(* Logix 5000 project; controller DispersionPlc vendor 1 type 14 code 108 rev 34.11; software revision 34.01 *)

TASK MainTask (continuous, watchdog 500 ms) : MainProgram, Unit_K400, Unit_V4307, Unit_V4306, Unit_T4302, Unit_S4352, Unit_S51, Unit_RO_HE4305, Simulation, General_Purpose, Deviation_Alarms, Unit_K200
TASK Periodic_100ms (periodic, rate 100 ms, priority 2, watchdog 500 ms) : PIDLoops

MODULES
   Local : vendor 1 type 14 code 108 (Compact 0, rev 34.11)
      Input_2 : vendor 1 type 7 code 82 (Compact 3, rev 1.1, Input RPI 2 ms)
      Input_1 : vendor 1 type 7 code 82 (Compact 2, rev 1.1, Input RPI 2 ms)
      Input_3 : vendor 1 type 7 code 82 (Compact 4, rev 1.1, Input RPI 2 ms)
      Therm_1 : vendor 1 type 10 code 36 (Compact 8, rev 1.2, Input RPI 2 ms)
      IF81 : 1769-MODULE (Compact 12, rev 1.1, Output RPI 2 ms)
      AnaOut : vendor 1 type 10 code 40 (Compact 13, rev 2.1, Output RPI 2 ms)
      Therm_3 : vendor 1 type 10 code 36 (Compact 10, rev 1.2, Input RPI 2 ms)
      Sdn : vendor 1 type 12 code 105 (Compact 1, rev 2.1, Output RPI 2 ms)
      IF8 : 1769-MODULE (Compact 11, rev 1.1, Output RPI 2 ms)
      Output_1 : 1769-OW16 (Compact 5, rev 1.1, Output RPI 2 ms)
      Output_2 : 1769-OW16 (Compact 6, rev 1.1, Output RPI 2 ms)
      Output_3 : 1769-OW16 (Compact 7, rev 1.1, Output RPI 2 ms)
      Therm_2 : vendor 1 type 10 code 36 (Compact 9, rev 1.2, Input RPI 2 ms)
      AG_4306 : PowerFlex 525-EENET (Ethernet 10.61.51.161, rev 5.1, Output RPI 20 ms)
      P_4302_2 : PowerFlex 525-EENET (Ethernet 10.61.51.163, rev 5.1, Output RPI 20 ms)
      AG_4302 : vendor 1 type 142 code 1168 (Ethernet 10.61.51.160, rev 9.1, Output RPI 20 ms)
          : vendor 1 type 142 code 57760 (RhinoBP 5, rev 1.1)
          : vendor 1 type 142 code 33184 (RhinoBP 14, rev 2.5)
      AG_4307 : PowerFlex 525-EENET (Ethernet 10.61.51.162, rev 5.1, Output RPI 20 ms)
      New_INX_IO : vendor 1 type 12 code 298 (Ethernet 10.61.51.115, rev 1.1)
         AC_Inputs : vendor 1 type 7 code 82 (Compact 1, rev 3.1, Input RPI 100 ms)
         Digital_Inputs : 1769-IQ16 (Compact 5, rev 1.1, Input RPI 20 ms)
         Relay_Outputs : 1769-OW8I (Compact 2, rev 3.1, Output RPI 100 ms)
         Analog_Inputs : vendor 1 type 10 code 44 (Compact 3, rev 2.1, Output RPI 100 ms)
         Analog_Outputs : vendor 1 type 10 code 40 (Compact 4, rev 2.2, Output RPI 100 ms)
         Digital_Outputs : 1769-OB16 (Compact 6, rev 2.1, Output RPI 20 ms)
      RIO1_Rack1 : vendor 1 type 12 code 298 (Ethernet 10.61.51.164, rev 1.1)
         DIn : vendor 1 type 7 code 82 (Compact 3, rev 1.1, Input RPI 20 ms)
         DOut : 1769-OW16 (Compact 4, rev 1.1, Output RPI 20 ms)
         AOut : vendor 1 type 10 code 40 (Compact 2, rev 2.1, Output RPI 80 ms)
         AIn : 1769-IF8 (Compact 1, rev 1.1, Output RPI 80 ms)
END_MODULES

TYPE Alarm_SPT :
STRUCT
   HIHI : REAL;
   HI : REAL;
   LO : REAL;
   LOLO : REAL;
END_STRUCT
END_TYPE

TYPE AStd_AnalogAlarm :
STRUCT
   AckC : BOOL;
   LatchA : BOOL;
   DetectS : BOOL;
   BitS : BOOL;
   InhibitC : BOOL;
   LimitC : REAL;
   LimitOffSetC : REAL;
   Tmr : TIMER;
   Disabled : BOOL;
END_STRUCT
END_TYPE

TYPE AStd_AnalogInput :
STRUCT
   Raw : REAL;
   AckAreaC : BOOL;
   AckC : BOOL;
   Scaled : REAL;
   Scaling : AStd_AnalogScaling;
   LowLow : AStd_AnalogAlarm;
   Low : AStd_AnalogAlarm;
   High : AStd_AnalogAlarm;
   HighHigh : AStd_AnalogAlarm;
   Fault : AStd_AnalogAlarm;
   FaultReset : REAL;
END_STRUCT
END_TYPE

TYPE AStd_AnalogOutput :
STRUCT
   Scaled : REAL;
   Raw : REAL;
   Scaling : AStd_AnalogScaling;
END_STRUCT
END_TYPE

TYPE AStd_AnalogScaling :
STRUCT
   RawMinS : REAL;
   RawMaxS : REAL;
   EngMinS : REAL;
   EngMaxS : REAL;
END_STRUCT
END_TYPE

TYPE AStd_DateTimeFormat :
STRUCT
   CurrentYear : DINT;
   CurrentMonth : DINT;
   CurrentDay : DINT;
   CurrentHour : DINT;
   CurrentMinute : DINT;
   CurrentSecond : DINT;
   DateTimeBuild : STRING;
   TemporaryString : STRING;
   DateTimeBuffer : DINT[10];
   ConstantZero : STRING;
   ConstantColon : STRING;
   ConstantDash : STRING;
   ConstantSpace : STRING;
   CurrentDateTime : STRING;
   SetTimeC : BOOL;
END_STRUCT
END_TYPE

TYPE AStd_Device_Perm :
STRUCT
   InterlockS : DINT;
   SafetyS : DINT;
   IntlkS : BOOL;
   SafeS : BOOL;
   InterlockInhibitC : DINT;
   SafetyInhibitC : DINT;
   IntSafDisp : DINT;
   InterlockTimers : TimerArray;
END_STRUCT
END_TYPE

TYPE AStd_DiscreteAlarm :
STRUCT
   AckC : BOOL;
   LatchA : BOOL;
   DetectS : BOOL;
   BitS : BOOL;
   InhibitC : BOOL;
   Tmr : TIMER;
END_STRUCT
END_TYPE

TYPE AStd_DiscreteInput :
STRUCT
   InI : BOOL;
   Alm : AStd_DiscreteAlarm;
END_STRUCT
END_TYPE

TYPE AStd_FVNR :
STRUCT
   AutoC : BOOL;
   ManC : BOOL;
   AutoS : BOOL;
   StartC : BOOL;
   StopC : BOOL;
   RunO : BOOL;
   RunI : BOOL;
   DiscI : BOOL;
   AlmS : BOOL;
   RuntimeResetC : BOOL;
   AutoCtrlS : BOOL;
   AutoCtrlC : DINT;
   RuntimeS : DINT;
   Perm : AStd_Device_Perm;
   MiscAlm : AStd_DiscreteAlarm;
   DiscAlm : AStd_DiscreteAlarm;
   AckC : BOOL;
END_STRUCT
END_TYPE

TYPE AStd_GeneralPurp :
STRUCT
   AlwaysOff : BOOL;
   AlwaysOn : BOOL;
   FirstScan : BOOL;
   PowerUpDelay : BOOL;
   AlternateScan : BOOL;
   HalfSecondPulse : BOOL;
   HalfSecondSquare : BOOL;
   OneSecondPulse : BOOL;
   OneSecondSquare : BOOL;
   PowerUpDelayOS : BOOL;
   Tmr : TIMER[5];
   ONS : DINT;
END_STRUCT
END_TYPE

TYPE AStd_PIDInterface :
STRUCT
   AutoC : BOOL;
   ManC : BOOL;
   AutoS : BOOL;
   AutoCtrlC : DINT;
   AutoCtrlS : BOOL;
   EnableS : BOOL;
   ManOut : REAL;
   SPC : REAL;
   PGainC : REAL;
   IGainC : REAL;
   DGainC : REAL;
   PGainS : REAL;
   IGainS : REAL;
   DGainS : REAL;
   SPS : REAL;
   PVS : REAL;
   CVS : REAL;
   Perm : AStd_Device_Perm;
END_STRUCT
END_TYPE

TYPE AStd_PLCStatus :
STRUCT
   ForcePresent : BOOL;
   BatteryFault : BOOL;
   MinorFaultBits : DINT;
   ForceStatus : DINT;
   PLCScanTime : REAL;
   PLCScanTimeMin : REAL;
   CodeVersion : STRING;
   DateTime : AStd_DateTimeFormat;
   PLCForcePresent : AStd_DiscreteAlarm;
   PLCBatteryFault : AStd_DiscreteAlarm;
   PLCPowerUp : AStd_DiscreteAlarm;
END_STRUCT
END_TYPE

TYPE AStd_PLI :
STRUCT
   StartC : BOOL;
   HoldC : BOOL;
   RestartC : BOOL;
   AbortC : BOOL;
   CompleteC : BOOL;
   ResetC : BOOL;
   UserStopC : BOOL;
   IdleS : BOOL;
   RunS : BOOL;
   HeldS : BOOL;
   AbortS : BOOL;
   DoneS : BOOL;
   CurrentStateCodeS : DINT;
   PreventStartS : DINT;
   AlarmS : DINT;
   Adv : BOOL;
   StepNo : DINT;
   StepBit : DINT;
   ONS : DINT;
   UnitProc_ActiveS : BOOL;
   UnitProc_RecipePointerS : DINT;
   UnitProc_PhaseID : DINT;
   RealParameters : REAL[20];
   BoolParameters : BOOL[32];
   DINTParameters : DINT[20];
   PreventStartInhibitC : DINT;
   AlarmInhibitC : DINT;
   IntSafDisp : DINT;
   InterlockTimers : TimerArray;
END_STRUCT
END_TYPE

TYPE AStd_VFD :
STRUCT
   AutoC : BOOL;
   ManC : BOOL;
   AutoS : BOOL;
   StartC : BOOL;
   StartRevC : BOOL;
   StopC : BOOL;
   ManSpdC : REAL;
   AutoSpdC : REAL[10];
   AutoSpdS : REAL;
   SpeedI : AStd_AnalogInput;
   SpeedC : AStd_AnalogOutput;
   AutoCtrlC : DINT;
   AutoRevCtrlC : DINT;
   AutoCtrlS : BOOL;
   AutoRevCtrlS : BOOL;
   RunI : BOOL;
   DiscI : BOOL;
   DriveFltI : BOOL;
   RunTimeResetC : BOOL;
   RunTimeS : DINT;
   RunO : BOOL;
   ReverseS : BOOL;
   AckC : BOOL;
   AckAreaC : BOOL;
   Perm : AStd_Device_Perm;
   MiscAlm : AStd_DiscreteAlarm;
   DiscAlm : AStd_DiscreteAlarm;
   DriveFlt : AStd_DiscreteAlarm;
   AlmS : BOOL;
END_STRUCT
END_TYPE

TYPE AStd_VlvModulating :
STRUCT
   AutoC : BOOL;
   ManC : BOOL;
   AutoS : BOOL;
   OpenC : BOOL;
   CloseC : BOOL;
   AutoCtrlS : BOOL;
   Perm : AStd_Device_Perm;
   ManPosC : REAL;
   AutoCtrlC : DINT;
   AutoPosC : REAL[10];
   AutoPosS : REAL;
   ScaledO : REAL;
   Scaling : AStd_AnalogScaling;
   RawO : REAL;
END_STRUCT
END_TYPE

TYPE AStd_VlvOC :
STRUCT
   AutoC : BOOL;
   ManC : BOOL;
   AutoS : BOOL;
   OpenC : BOOL;
   CloseC : BOOL;
   StopC : BOOL;
   OpenO : BOOL;
   CloseO : BOOL;
   OpenI : BOOL;
   ClosedI : BOOL;
   CycleCountResetC : BOOL;
   AlmS : BOOL;
   AutoCtrlS : BOOL;
   AckC : BOOL;
   AckAreaC : BOOL;
   cfgHasZSC : BOOL;
   cfgHasZSO : BOOL;
   AutoCtrlC : DINT;
   CycleCountS : DINT;
   Perm : AStd_Device_Perm;
   MiscAlm : AStd_DiscreteAlarm;
END_STRUCT
END_TYPE

TYPE bit64 :
STRUCT
   Bit : BOOL[64];
END_STRUCT
END_TYPE

TYPE Kettle :
STRUCT
   Level : Proc_Var;
   Heating : Proc_Var;
   Pressure : Proc_Var;
   Cooling : Proc_Var;
   Combined : Proc_Var;
   Auto_Manual : BOOL;
   Heat_Manual_Output_Request : REAL;
   ValveOutput : INT;
   CoolingValveOutput : INT;
   ValvePercOpen : REAL;
   OverheadTemp : REAL;
   H20SupplyValvePercOpen : REAL;
   H20SupplyValveOutput : INT;
   RupDiscRelfTemp : REAL;
   Zone1ActuatedValvePos : BOOL;
   Zone2ActuatedValvePos : BOOL;
   Zone3ActuatedValvePos : BOOL;
   Cool_Auto_Manual : BOOL;
   Cool_Manual_Output_Request : REAL;
   BatchStart : BOOL;
   BatchRunning : BOOL;
   BatchID : STRING;
   ProductID : STRING;
   Proportional : REAL;
   Integral : REAL;
   Derivative : REAL;
   Timer : TIMER[5];
   BatchStop : BOOL;
   Alarm : BOOL;
   Cooling_Valve_Status : BOOL;
   Reflux : BOOL;
   BIts : DINT;
   Operation : DINT;
END_STRUCT
END_TYPE

TYPE Proc_Var :
STRUCT
   Value_Name : STRING;
   Value_Raw : INT;
   Value : REAL;
   Volume_Value : REAL;
   Setpoint : REAL;
   Error_Val : REAL;
   MMI_Level : REAL;
   Value_Sf : REAL;
   Volume_Sf : REAL;
   Offset : REAL;
   HIHI : REAL;
   HI : REAL;
   LO : REAL;
   LOLO : REAL;
   OUT : REAL;
   HIHI_ALM : BOOL;
   HI_ALM : BOOL;
   LO_ALM : BOOL;
   LOLO_ALM : BOOL;
   High_Limit_Switch : BOOL;
   Lo_Limit_Switch : BOOL;
   LossOfInput : BOOL;
END_STRUCT
END_TYPE

TYPE Seq64 :
STRUCT
   Val : DINT;
   Ret : DINT;
   Tmr : TIMER[64];
   probit : BOOL[64];
   Ons : BOOL[64];
   seqstrings : STRING[64];
   alarmstrings : STRING[64];
   seqstring : STRING;
   alarmstring : STRING;
   Alarm_Timers : TIMER[64];
   Alarm_Scanner : DINT;
   Alarm_Display_Index : DINT;
   Alarm_Display_Que : DINT;
   ClearAlarms : BOOL;
   Active : BOOL;
   Sq : Stp64;
   MANUAL : bit64;
   Alarm : bit64;
   ALARM_TIMER : TIMER;
   ALARM_DISPLAY : DINT;
   AutoMode : BOOL;
   ManualMode : BOOL;
   AutoManualPb : BOOL;
   ClearAlarmTmr : TIMER;
   HMI : bit64;
   VAL_HOLD : DINT;
   CLEAR_SEQ : BOOL;
   AlarmHist : bit64;
   AlarmHistEnable : bit64;
   AlarmONS : bit64;
   AlarmHistString : STRING;
   Alarm_Setpoint : Alarm_SPT;
END_STRUCT
END_TYPE

TYPE Stp64 :
STRUCT
   Step : BOOL[64];
   Dn : BOOL[64];
END_STRUCT
END_TYPE

TYPE TimerArray :
STRUCT
   Timers : TIMER[10];
END_STRUCT
END_TYPE

TYPE Udt_Tank :
STRUCT
   Name : STRING;
   Level : Proc_Var;
   Temperature : Proc_Var;
   Pressure : Proc_Var;
   PercentChange : REAL;
   MaxPercentChange : BOOL;
   LvlSampleAtPmpStart : REAL;
   Enabled : BOOL;
   MaxPercChangeAlr : BOOL;
   Number : INT;
END_STRUCT
END_TYPE

TYPE VFD :
STRUCT
   TargetDriveSpeed : INT;
   I_Ready : BOOL;
   I_Running : BOOL;
   I_CmdDir : BOOL;
   I_ActDir : BOOL;
   I_Accelerating : BOOL;
   I_Decelerating : BOOL;
   I_Alarm : BOOL;
   I_Fault : BOOL;
   I_AtSpeed : BOOL;
   I_LocalContStat1 : BOOL;
   I_LocalContStat2 : BOOL;
   I_LocalContStat3 : BOOL;
   I_Refferance1 : BOOL;
   I_Refferance2 : BOOL;
   I_Refferance3 : BOOL;
   I_Refferance4 : BOOL;
   I_V_Units_Fb : REAL;
   I_Act_Amps : REAL;
   I_DatalinkA2_Fb : REAL;
   O_Stop : BOOL;
   O_Run : BOOL;
   O_Jog : BOOL;
   O_ClrFlts : BOOL;
   O_DirBit1 : BOOL;
   O_DirBit2 : BOOL;
   O_LocalContol : BOOL;
   O_MopInc : BOOL;
   O_MOP_Accel1 : BOOL;
   O_Accel2 : BOOL;
   O_MOP_Decel1 : BOOL;
   O_MOP_Decel2 : BOOL;
   O_Reff_Sel1 : BOOL;
   O_Reff_Sel2 : BOOL;
   O_Reff_Sel3 : BOOL;
   O_V_CmdReff : REAL;
   O_Dlnk_A1_Reff : INT;
   O_Dlnk_A2_Reff : INT;
   SpeedScaleIn : REAL;
   SpeedScaleOut : REAL;
   MaxOutPut : REAL;
   MinOutput : REAL;
   DriveSpeedReff : REAL;
END_STRUCT
END_TYPE

ADD_ON_INSTRUCTION Analog_Scale   (* revision 1.0, vendor DM *)
VAR_INPUT
   Analog_In : REAL; {required}
   Offset_In : REAL; {required}
   Analog_Min_In : REAL; {required}
   Analog_Max_In : REAL; {required}
   Analog_Min_Out : REAL; {required}
   Analog_Max_Out : REAL; {required}
END_VAR
VAR_OUTPUT
   Analog_Out : REAL; {access Read Only, required}
END_VAR
VAR_INPUT
   Offset_Out : REAL; {required}
END_VAR
VAR
   F8 : REAL[10];
END_VAR

ROUTINE Logic   (* ladder *)
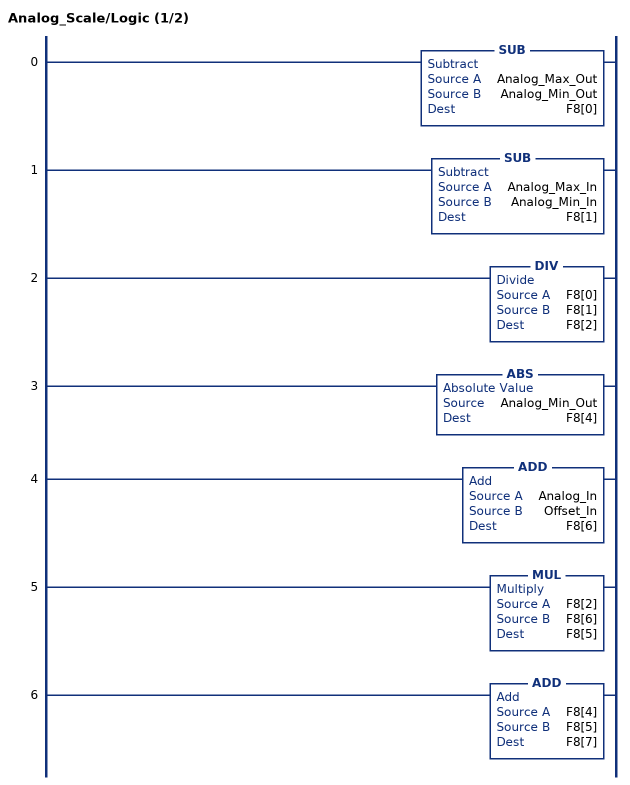
   0: SUB(Analog_Max_Out,Analog_Min_Out,F8[0]);
   1: SUB(Analog_Max_In,Analog_Min_In,F8[1]);
   2: DIV(F8[0],F8[1],F8[2]);
   3: ABS(Analog_Min_Out,F8[4]);
   4: ADD(Analog_In,Offset_In,F8[6]);
   5: MUL(F8[2],F8[6],F8[5]);
   6: ADD(F8[4],F8[5],F8[7]);
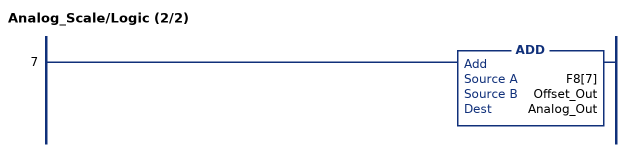
   7: ADD(F8[7],Offset_Out,Analog_Out);
END_ROUTINE
END_ADD_ON_INSTRUCTION

ADD_ON_INSTRUCTION AOI_Toggle   (* revision 1.0, vendor Danieli Taranis, ExecutePrescan, ExecuteEnableInFalse *)
VAR_OUTPUT
   Q : BOOL; {visible}
   QNot : BOOL; {visible}
END_VAR
VAR
   StorageBit : BOOL; {access None}
   RunOnce : BOOL; {access None}
END_VAR

ROUTINE EnableInFalse   (* structured text *)
   RunOnce:=0;
END_ROUTINE

ROUTINE Logic   (* structured text *)
   //Perform one shot logic and
   //then evaluate the state of Q.
   //
   //Flip value of Q to opposite value.
   //Set QNot to opposite of Q
   //Store internal RunOnce for one shot logic
   
   IF NOT RunOnce THEN
   
   	Q:=NOT Q;
   	QNot:=NOT Q;
   	RunOnce:=1;
   
   END_IF;
   
   
   
   
END_ROUTINE

ROUTINE Prescan   (* structured text *)
   Q:=0;
   RunOnce:=0;
   
END_ROUTINE
END_ADD_ON_INSTRUCTION

ADD_ON_INSTRUCTION AStd_AI_AOI   (* revision 1.0, vendor Avanceon *)
VAR_IN_OUT
   AnalogInput : AStd_AnalogInput; {required}
END_VAR
VAR_INPUT
   InputRaw_I : REAL; {required}
   cfgRawMin : REAL := 4000.0; {required}
   cfgRawMax : REAL := 20000.0; {required}
   cfgEUMin : REAL; {required}
   cfgEUMax : REAL := 100.0; {required}
END_VAR
VAR_OUTPUT
   Scaled : REAL; {access Read Only, visible}
END_VAR
VAR_INPUT
   CommsStatus : BOOL; {required}
END_VAR

ROUTINE Logic   (* ladder *)
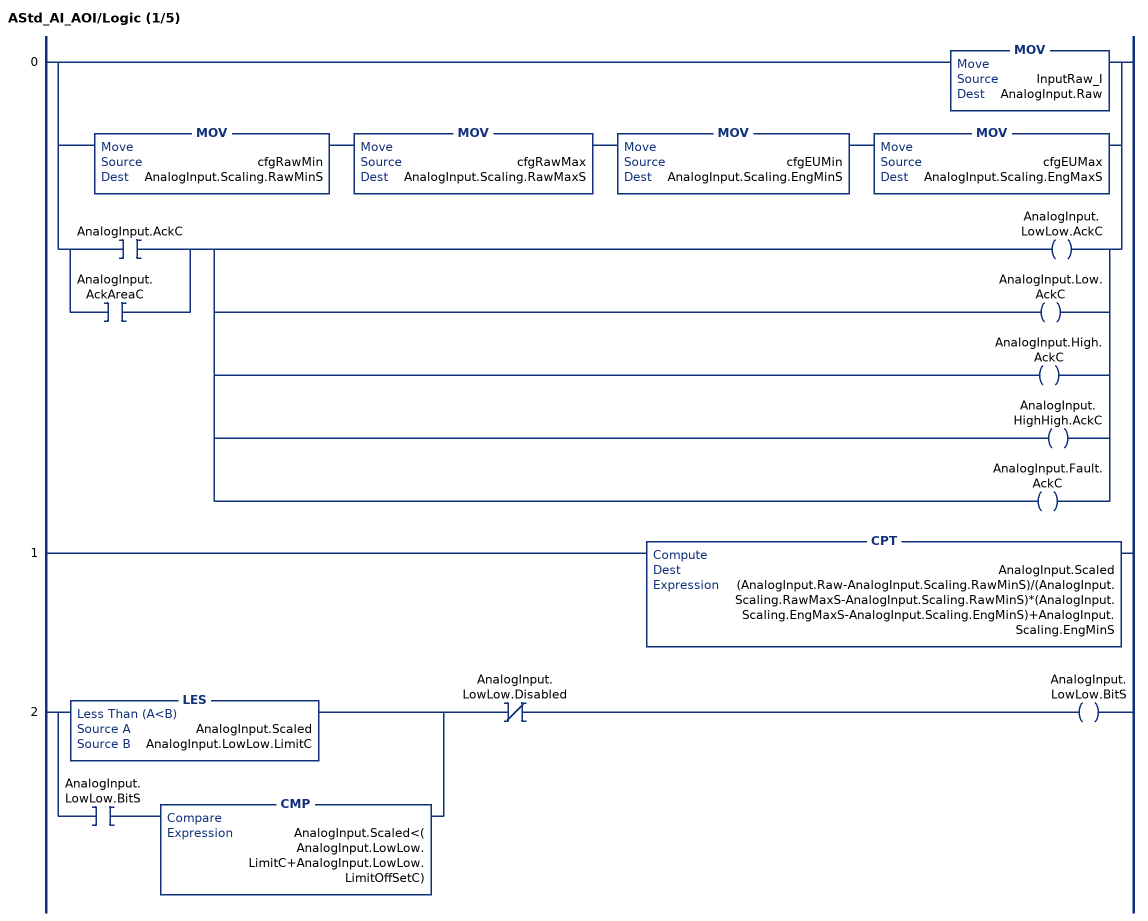
   0: [MOV(InputRaw_I,AnalogInput.Raw) ,MOV(cfgRawMin,AnalogInput.Scaling.RawMinS) MOV(cfgRawMax,AnalogInput.Scaling.RawMaxS) MOV(cfgEUMin,AnalogInput.Scaling.EngMinS) MOV(cfgEUMax,AnalogInput.Scaling.EngMaxS) ,[XIC(AnalogInput.AckC) ,XIC(AnalogInput.AckAreaC) ] [OTE(AnalogInput.LowLow.AckC) ,OTE(AnalogInput.Low.AckC) ,OTE(AnalogInput.High.AckC) ,OTE(AnalogInput.HighHigh.AckC) ,OTE(AnalogInput.Fault.AckC) ] ];
   1: CPT(AnalogInput.Scaled,(AnalogInput.Raw-AnalogInput.Scaling.RawMinS)/(AnalogInput.Scaling.RawMaxS-AnalogInput.Scaling.RawMinS)*(AnalogInput.Scaling.EngMaxS-AnalogInput.Scaling.EngMinS)+AnalogInput.Scaling.EngMinS);
   2: [LES(AnalogInput.Scaled,AnalogInput.LowLow.LimitC) ,XIC(AnalogInput.LowLow.BitS) CMP(AnalogInput.Scaled<(AnalogInput.LowLow.LimitC+AnalogInput.LowLow.LimitOffSetC)) ]XIO(AnalogInput.LowLow.Disabled)OTE(AnalogInput.LowLow.BitS);
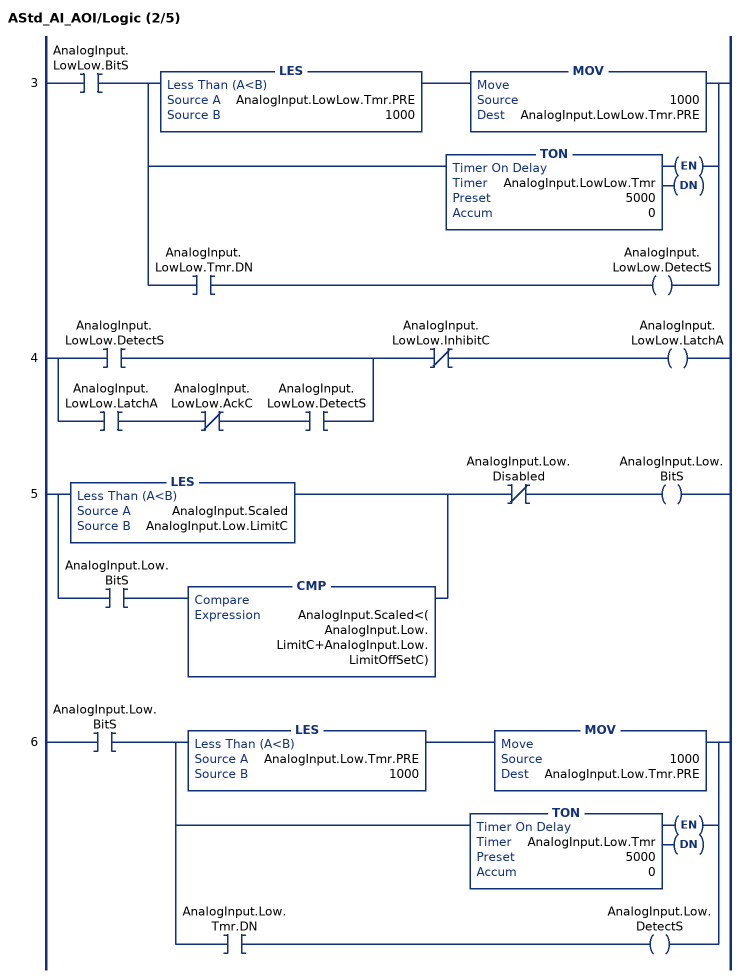
   3: XIC(AnalogInput.LowLow.BitS)[LES(AnalogInput.LowLow.Tmr.PRE,1000) MOV(1000,AnalogInput.LowLow.Tmr.PRE) ,TON(AnalogInput.LowLow.Tmr,5000,0) ,XIC(AnalogInput.LowLow.Tmr.DN) OTE(AnalogInput.LowLow.DetectS) ];
   4: [XIC(AnalogInput.LowLow.DetectS) ,XIC(AnalogInput.LowLow.LatchA) XIO(AnalogInput.LowLow.AckC) XIC(AnalogInput.LowLow.DetectS) ]XIO(AnalogInput.LowLow.InhibitC)OTE(AnalogInput.LowLow.LatchA);
   5: [LES(AnalogInput.Scaled,AnalogInput.Low.LimitC) ,XIC(AnalogInput.Low.BitS) CMP(AnalogInput.Scaled<(AnalogInput.Low.LimitC+AnalogInput.Low.LimitOffSetC)) ]XIO(AnalogInput.Low.Disabled)OTE(AnalogInput.Low.BitS);
   6: XIC(AnalogInput.Low.BitS)[LES(AnalogInput.Low.Tmr.PRE,1000) MOV(1000,AnalogInput.Low.Tmr.PRE) ,TON(AnalogInput.Low.Tmr,5000,0) ,XIC(AnalogInput.Low.Tmr.DN) OTE(AnalogInput.Low.DetectS) ];
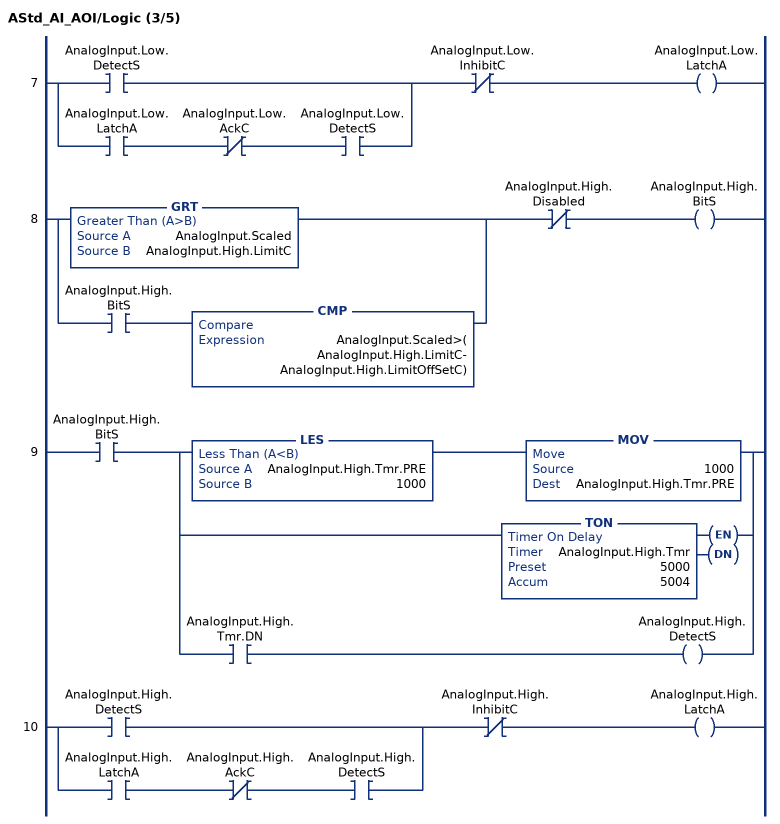
   7: [XIC(AnalogInput.Low.DetectS) ,XIC(AnalogInput.Low.LatchA) XIO(AnalogInput.Low.AckC) XIC(AnalogInput.Low.DetectS) ]XIO(AnalogInput.Low.InhibitC)OTE(AnalogInput.Low.LatchA);
   8: [GRT(AnalogInput.Scaled,AnalogInput.High.LimitC) ,XIC(AnalogInput.High.BitS) CMP(AnalogInput.Scaled>(AnalogInput.High.LimitC-AnalogInput.High.LimitOffSetC)) ]XIO(AnalogInput.High.Disabled)OTE(AnalogInput.High.BitS);
   9: XIC(AnalogInput.High.BitS)[LES(AnalogInput.High.Tmr.PRE,1000) MOV(1000,AnalogInput.High.Tmr.PRE) ,TON(AnalogInput.High.Tmr,5000,5004) ,XIC(AnalogInput.High.Tmr.DN) OTE(AnalogInput.High.DetectS) ];
   10: [XIC(AnalogInput.High.DetectS) ,XIC(AnalogInput.High.LatchA) XIO(AnalogInput.High.AckC) XIC(AnalogInput.High.DetectS) ]XIO(AnalogInput.High.InhibitC)OTE(AnalogInput.High.LatchA);
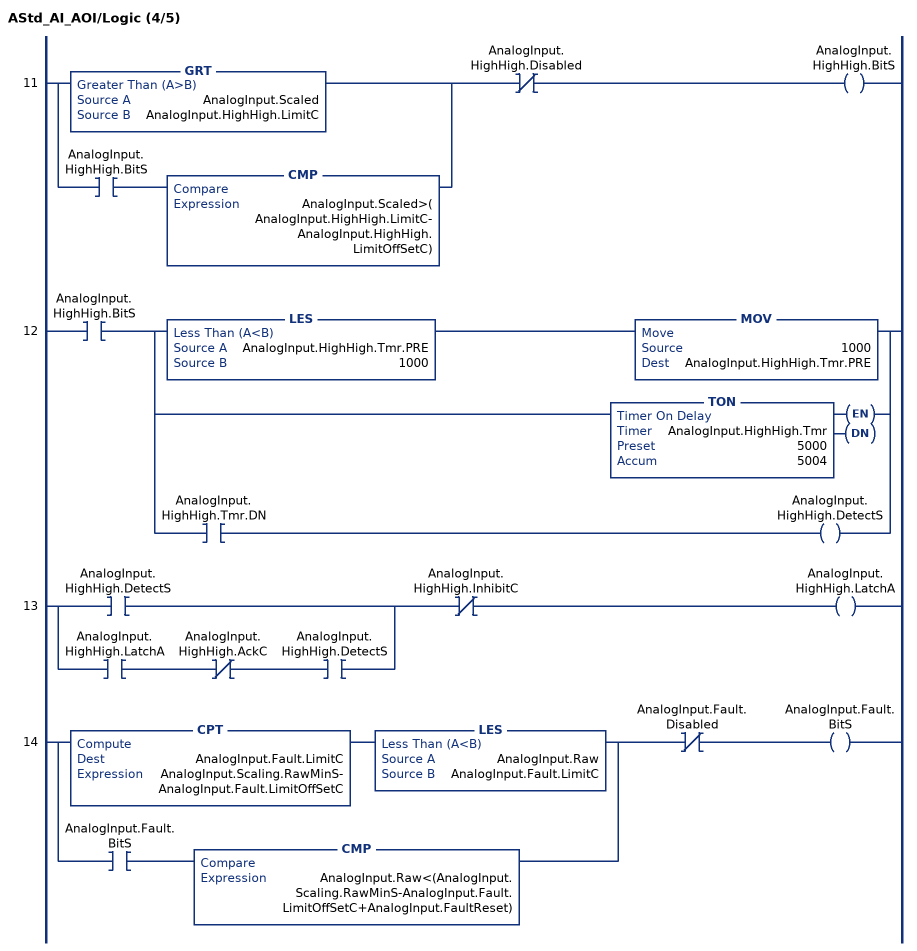
   11: [GRT(AnalogInput.Scaled,AnalogInput.HighHigh.LimitC) ,XIC(AnalogInput.HighHigh.BitS) CMP(AnalogInput.Scaled>(AnalogInput.HighHigh.LimitC-AnalogInput.HighHigh.LimitOffSetC)) ]XIO(AnalogInput.HighHigh.Disabled)OTE(AnalogInput.HighHigh.BitS);
   12: XIC(AnalogInput.HighHigh.BitS)[LES(AnalogInput.HighHigh.Tmr.PRE,1000) MOV(1000,AnalogInput.HighHigh.Tmr.PRE) ,TON(AnalogInput.HighHigh.Tmr,5000,5004) ,XIC(AnalogInput.HighHigh.Tmr.DN) OTE(AnalogInput.HighHigh.DetectS) ];
   13: [XIC(AnalogInput.HighHigh.DetectS) ,XIC(AnalogInput.HighHigh.LatchA) XIO(AnalogInput.HighHigh.AckC) XIC(AnalogInput.HighHigh.DetectS) ]XIO(AnalogInput.HighHigh.InhibitC)OTE(AnalogInput.HighHigh.LatchA);
   14: [CPT(AnalogInput.Fault.LimitC,AnalogInput.Scaling.RawMinS-AnalogInput.Fault.LimitOffSetC) LES(AnalogInput.Raw,AnalogInput.Fault.LimitC) ,XIC(AnalogInput.Fault.BitS) CMP(AnalogInput.Raw<(AnalogInput.Scaling.RawMinS-AnalogInput.Fault.LimitOffSetC+AnalogInput.FaultReset)) ]XIO(AnalogInput.Fault.Disabled)OTE(AnalogInput.Fault.BitS);
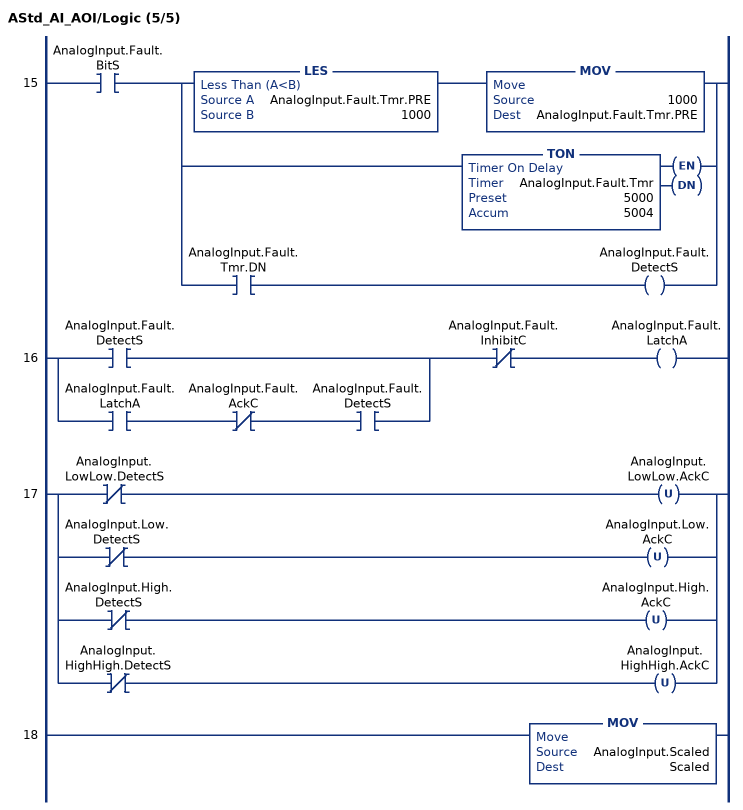
   15: XIC(AnalogInput.Fault.BitS)[LES(AnalogInput.Fault.Tmr.PRE,1000) MOV(1000,AnalogInput.Fault.Tmr.PRE) ,TON(AnalogInput.Fault.Tmr,5000,5004) ,XIC(AnalogInput.Fault.Tmr.DN) OTE(AnalogInput.Fault.DetectS) ];
   16: [XIC(AnalogInput.Fault.DetectS) ,XIC(AnalogInput.Fault.LatchA) XIO(AnalogInput.Fault.AckC) XIC(AnalogInput.Fault.DetectS) ]XIO(AnalogInput.Fault.InhibitC)OTE(AnalogInput.Fault.LatchA);
   17: [XIO(AnalogInput.LowLow.DetectS) OTU(AnalogInput.LowLow.AckC) ,XIO(AnalogInput.Low.DetectS) OTU(AnalogInput.Low.AckC) ,XIO(AnalogInput.High.DetectS) OTU(AnalogInput.High.AckC) ,XIO(AnalogInput.HighHigh.DetectS) OTU(AnalogInput.HighHigh.AckC) ];
   18: MOV(AnalogInput.Scaled,Scaled);
END_ROUTINE
END_ADD_ON_INSTRUCTION

ADD_ON_INSTRUCTION AStd_DI_AOI   (* revision 1.0, vendor Avanceon *)
VAR_IN_OUT
   DiscInputDevice : AStd_DiscreteInput; {required}
END_VAR
VAR_INPUT
   Input_I : BOOL; {access None, required}
   cfgFailSafe : BOOL; {access None, visible}
   cfgDebounceTmrPre : DINT := 1000; {access None, visible}
   cfgAlarmEnable : BOOL := 1; {access None, visible}
END_VAR
VAR_OUTPUT
   AlmS : BOOL; {access None, visible}
END_VAR
VAR
   Debounce : TIMER; {access None}
END_VAR

ROUTINE Logic   (* ladder *)
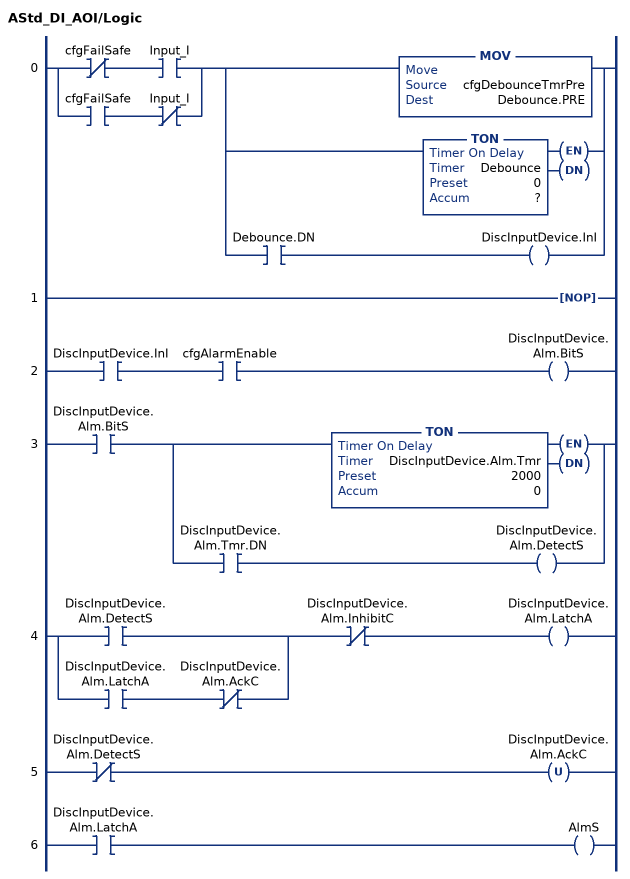
   0: [XIO(cfgFailSafe) XIC(Input_I) ,XIC(cfgFailSafe) XIO(Input_I) ][MOV(cfgDebounceTmrPre,Debounce.PRE) ,TON(Debounce,?,?) ,XIC(Debounce.DN) OTE(DiscInputDevice.InI) ];
   1: NOP();
   2: XIC(DiscInputDevice.InI)XIC(cfgAlarmEnable)OTE(DiscInputDevice.Alm.BitS);
   3: XIC(DiscInputDevice.Alm.BitS)[TON(DiscInputDevice.Alm.Tmr,2000,0) ,XIC(DiscInputDevice.Alm.Tmr.DN) OTE(DiscInputDevice.Alm.DetectS) ];
   4: [XIC(DiscInputDevice.Alm.DetectS) ,XIC(DiscInputDevice.Alm.LatchA) XIO(DiscInputDevice.Alm.AckC) ]XIO(DiscInputDevice.Alm.InhibitC)OTE(DiscInputDevice.Alm.LatchA);
   5: XIO(DiscInputDevice.Alm.DetectS)OTU(DiscInputDevice.Alm.AckC);
   6: XIC(DiscInputDevice.Alm.LatchA)OTE(AlmS);
END_ROUTINE
END_ADD_ON_INSTRUCTION

ADD_ON_INSTRUCTION AStd_FVNR_AOI   (* revision 1.0, vendor Avanceon *)
VAR_IN_OUT
   Motor : AStd_FVNR; {required}
END_VAR
VAR_INPUT
   AuxContact_I : BOOL; {required}
   Disconnect_I : BOOL; {required}
END_VAR
VAR_OUTPUT
   Coil_O : BOOL; {required}
END_VAR
VAR_INPUT
   cfgHasAUX : BOOL := 1; {access None, visible}
   cfgHasDISC : BOOL; {access None, visible}
END_VAR
VAR_OUTPUT
   AutoS : BOOL; {access Read Only, visible}
   RunS : BOOL; {access Read Only, visible}
   AlmS : BOOL; {access Read Only, visible}
END_VAR
VAR
   RuntimeHourTimer : TIMER := (PRE := 3600000); {access None}
END_VAR

ROUTINE Logic   (* ladder *)
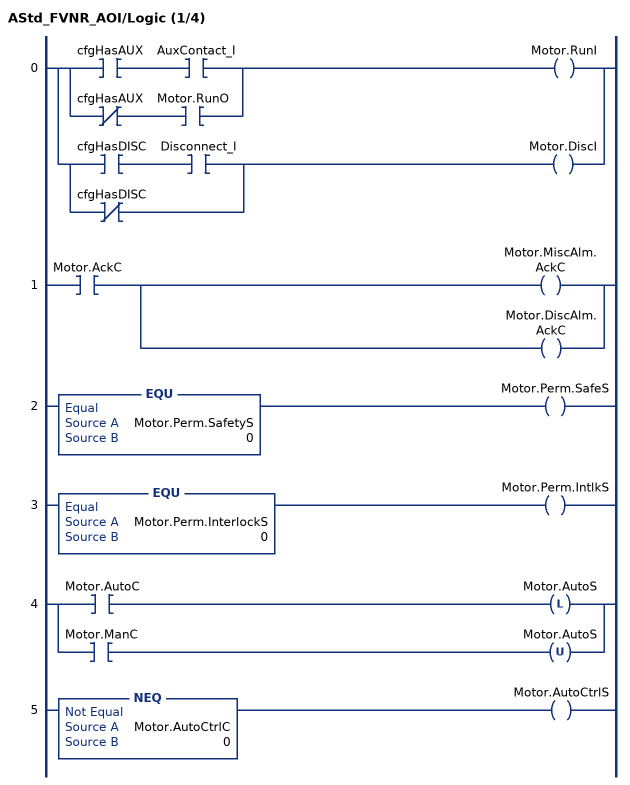
   0: [[XIC(cfgHasAUX) XIC(AuxContact_I) ,XIO(cfgHasAUX) XIC(Motor.RunO) ] OTE(Motor.RunI) ,[XIC(cfgHasDISC) XIC(Disconnect_I) ,XIO(cfgHasDISC) ] OTE(Motor.DiscI) ];
   1: XIC(Motor.AckC)[OTE(Motor.MiscAlm.AckC) ,OTE(Motor.DiscAlm.AckC) ];
   2: EQU(Motor.Perm.SafetyS,0)OTE(Motor.Perm.SafeS);
   3: EQU(Motor.Perm.InterlockS,0)OTE(Motor.Perm.IntlkS);
   4: [XIC(Motor.AutoC) OTL(Motor.AutoS) ,XIC(Motor.ManC) OTU(Motor.AutoS) ];
   5: NEQ(Motor.AutoCtrlC,0)OTE(Motor.AutoCtrlS);
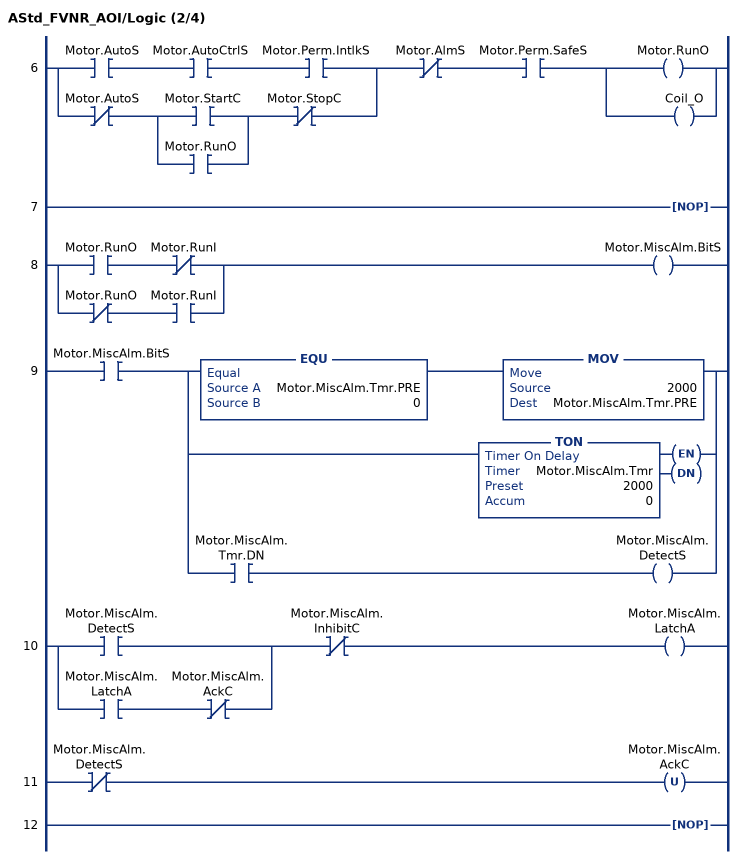
   6: [XIC(Motor.AutoS) XIC(Motor.AutoCtrlS) XIC(Motor.Perm.IntlkS) ,XIO(Motor.AutoS) [XIC(Motor.StartC) ,XIC(Motor.RunO) ] XIO(Motor.StopC) ]XIO(Motor.AlmS)XIC(Motor.Perm.SafeS)[OTE(Motor.RunO) ,OTE(Coil_O) ];
   7: NOP();
   8: [XIC(Motor.RunO) XIO(Motor.RunI) ,XIO(Motor.RunO) XIC(Motor.RunI) ]OTE(Motor.MiscAlm.BitS);
   9: XIC(Motor.MiscAlm.BitS)[EQU(Motor.MiscAlm.Tmr.PRE,0) MOV(2000,Motor.MiscAlm.Tmr.PRE) ,TON(Motor.MiscAlm.Tmr,2000,0) ,XIC(Motor.MiscAlm.Tmr.DN) OTE(Motor.MiscAlm.DetectS) ];
   10: [XIC(Motor.MiscAlm.DetectS) ,XIC(Motor.MiscAlm.LatchA) XIO(Motor.MiscAlm.AckC) ]XIO(Motor.MiscAlm.InhibitC)OTE(Motor.MiscAlm.LatchA);
   11: XIO(Motor.MiscAlm.DetectS)OTU(Motor.MiscAlm.AckC);
   12: NOP();
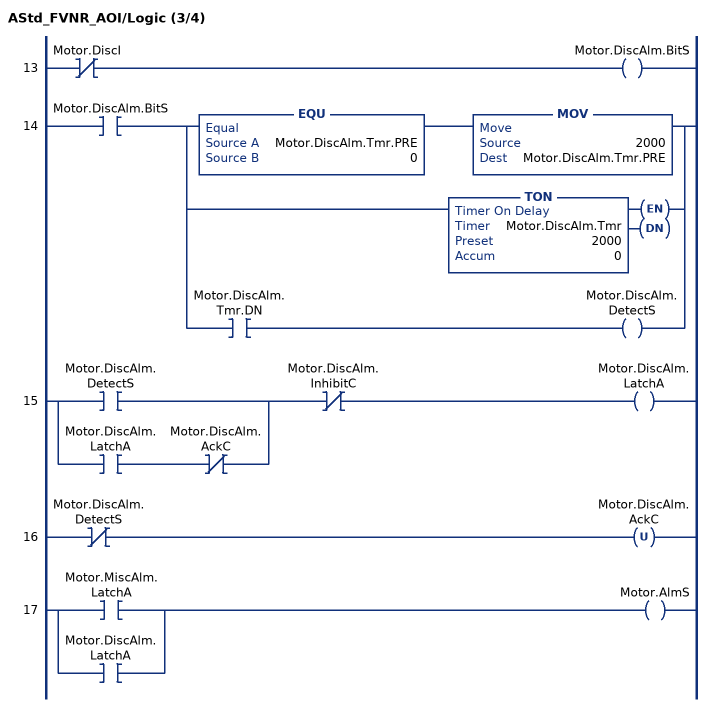
   13: XIO(Motor.DiscI)OTE(Motor.DiscAlm.BitS);
   14: XIC(Motor.DiscAlm.BitS)[EQU(Motor.DiscAlm.Tmr.PRE,0) MOV(2000,Motor.DiscAlm.Tmr.PRE) ,TON(Motor.DiscAlm.Tmr,2000,0) ,XIC(Motor.DiscAlm.Tmr.DN) OTE(Motor.DiscAlm.DetectS) ];
   15: [XIC(Motor.DiscAlm.DetectS) ,XIC(Motor.DiscAlm.LatchA) XIO(Motor.DiscAlm.AckC) ]XIO(Motor.DiscAlm.InhibitC)OTE(Motor.DiscAlm.LatchA);
   16: XIO(Motor.DiscAlm.DetectS)OTU(Motor.DiscAlm.AckC);
   17: [XIC(Motor.MiscAlm.LatchA) ,XIC(Motor.DiscAlm.LatchA) ]OTE(Motor.AlmS);
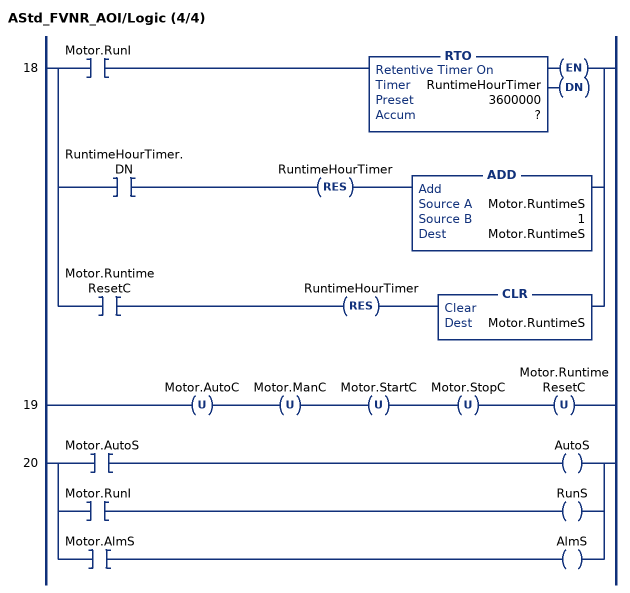
   18: [XIC(Motor.RunI) RTO(RuntimeHourTimer,?,?) ,XIC(RuntimeHourTimer.DN) RES(RuntimeHourTimer) ADD(Motor.RuntimeS,1,Motor.RuntimeS) ,XIC(Motor.RuntimeResetC) RES(RuntimeHourTimer) CLR(Motor.RuntimeS) ];
   19: OTU(Motor.AutoC)OTU(Motor.ManC)OTU(Motor.StartC)OTU(Motor.StopC)OTU(Motor.RuntimeResetC);
   20: [XIC(Motor.AutoS) OTE(AutoS) ,XIC(Motor.RunI) OTE(RunS) ,XIC(Motor.AlmS) OTE(AlmS) ];
END_ROUTINE
END_ADD_ON_INSTRUCTION

ADD_ON_INSTRUCTION AStd_PIDInterface_AOI   (* revision 1.0 *)
VAR_IN_OUT
   LoopInterface : AStd_PIDInterface; {required}
   PIDBlock : PID_ENHANCED; {required}
END_VAR
VAR_OUTPUT
   SP : REAL; {visible}
END_VAR
VAR_INPUT
   PV : REAL; {access Read Only, required}
END_VAR
VAR_OUTPUT
   CV : REAL; {access Read Only, required}
END_VAR
VAR_INPUT
   cfgCVSafeStatePCT : REAL; {access None, visible}
   cfgPVMinEU : REAL; {access None, visible}
   cfgPVMaxEU : REAL; {access None, visible}
END_VAR

ROUTINE Logic   (* ladder *)
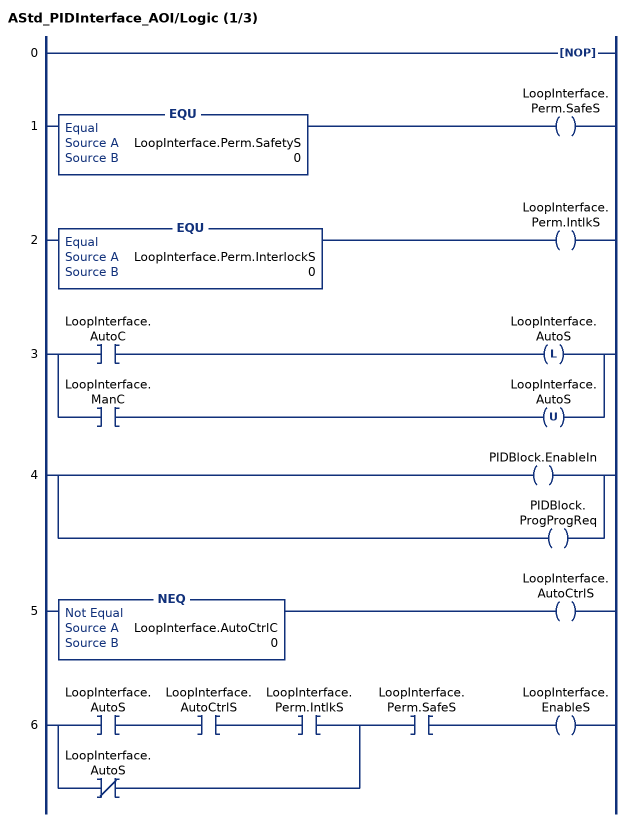
   0: NOP();
   1: EQU(LoopInterface.Perm.SafetyS,0)OTE(LoopInterface.Perm.SafeS);
   2: EQU(LoopInterface.Perm.InterlockS,0)OTE(LoopInterface.Perm.IntlkS);
   3: [XIC(LoopInterface.AutoC) OTL(LoopInterface.AutoS) ,XIC(LoopInterface.ManC) OTU(LoopInterface.AutoS) ];
   4: [OTE(PIDBlock.EnableIn) ,OTE(PIDBlock.ProgProgReq) ];
   5: NEQ(LoopInterface.AutoCtrlC,0)OTE(LoopInterface.AutoCtrlS);
   6: [XIC(LoopInterface.AutoS) XIC(LoopInterface.AutoCtrlS) XIC(LoopInterface.Perm.IntlkS) ,XIO(LoopInterface.AutoS) ]XIC(LoopInterface.Perm.SafeS)OTE(LoopInterface.EnableS);
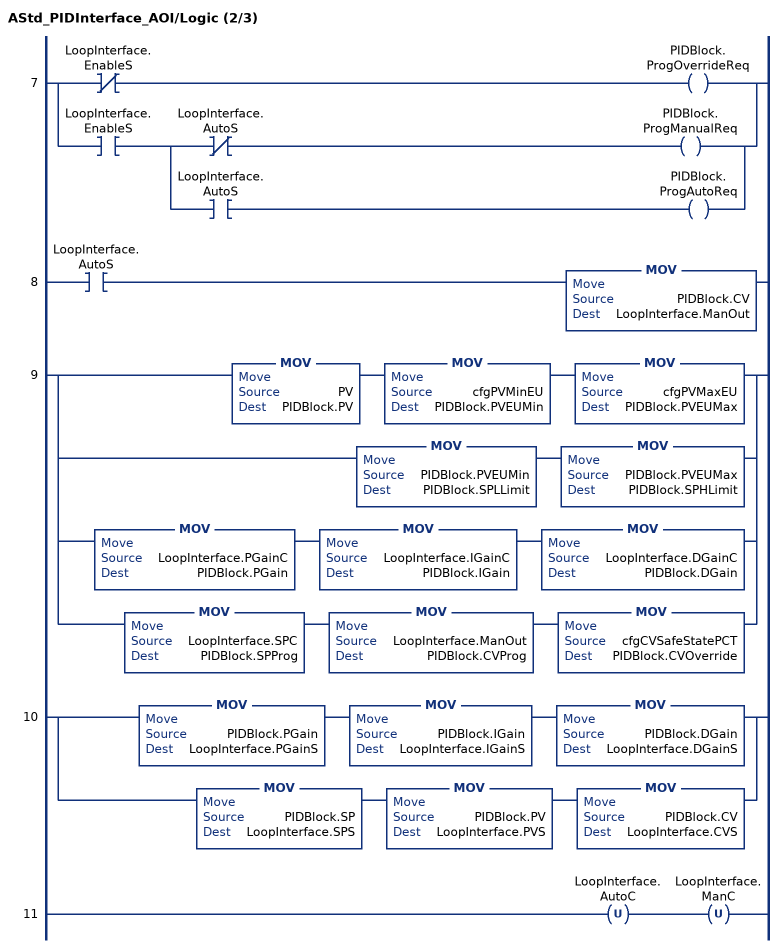
   7: [XIO(LoopInterface.EnableS) OTE(PIDBlock.ProgOverrideReq) ,XIC(LoopInterface.EnableS) [XIO(LoopInterface.AutoS) OTE(PIDBlock.ProgManualReq) ,XIC(LoopInterface.AutoS) OTE(PIDBlock.ProgAutoReq) ] ];
   8: XIC(LoopInterface.AutoS)MOV(PIDBlock.CV,LoopInterface.ManOut);
   9: [MOV(PV,PIDBlock.PV) MOV(cfgPVMinEU,PIDBlock.PVEUMin) MOV(cfgPVMaxEU,PIDBlock.PVEUMax) ,MOV(PIDBlock.PVEUMin,PIDBlock.SPLLimit) MOV(PIDBlock.PVEUMax,PIDBlock.SPHLimit) ,MOV(LoopInterface.PGainC,PIDBlock.PGain) MOV(LoopInterface.IGainC,PIDBlock.IGain) MOV(LoopInterface.DGainC,PIDBlock.DGain) ,MOV(LoopInterface.SPC,PIDBlock.SPProg) MOV(LoopInterface.ManOut,PIDBlock.CVProg) MOV(cfgCVSafeStatePCT,PIDBlock.CVOverride) ];
   10: [MOV(PIDBlock.PGain,LoopInterface.PGainS) MOV(PIDBlock.IGain,LoopInterface.IGainS) MOV(PIDBlock.DGain,LoopInterface.DGainS) ,MOV(PIDBlock.SP,LoopInterface.SPS) MOV(PIDBlock.PV,LoopInterface.PVS) MOV(PIDBlock.CV,LoopInterface.CVS) ];
   11: OTU(LoopInterface.AutoC)OTU(LoopInterface.ManC);
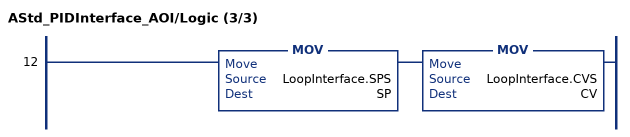
   12: MOV(LoopInterface.SPS,SP)MOV(LoopInterface.CVS,CV);
END_ROUTINE
END_ADD_ON_INSTRUCTION

ADD_ON_INSTRUCTION AStd_PLI_AOI   (* revision 0.0, vendor Avanceon *)
VAR_IN_OUT
   PLI : AStd_PLI; {required}
END_VAR
VAR_OUTPUT
   PreventStartS : BOOL; {access Read Only, visible}
   HeldS : BOOL; {access Read Only, visible}
   RunS : BOOL; {access Read Only, visible}
   AlmS : BOOL; {access Read Only, visible}
   StepNo : DINT; {access Read Only, visible}
END_VAR
VAR_INPUT
   cfgAutoReset : BOOL := 1; {visible}
   cfgPhaseID : DINT; {visible}
END_VAR
VAR
   AnyCmdActive : BOOL; {access None}
END_VAR

ROUTINE Logic   (* ladder *)
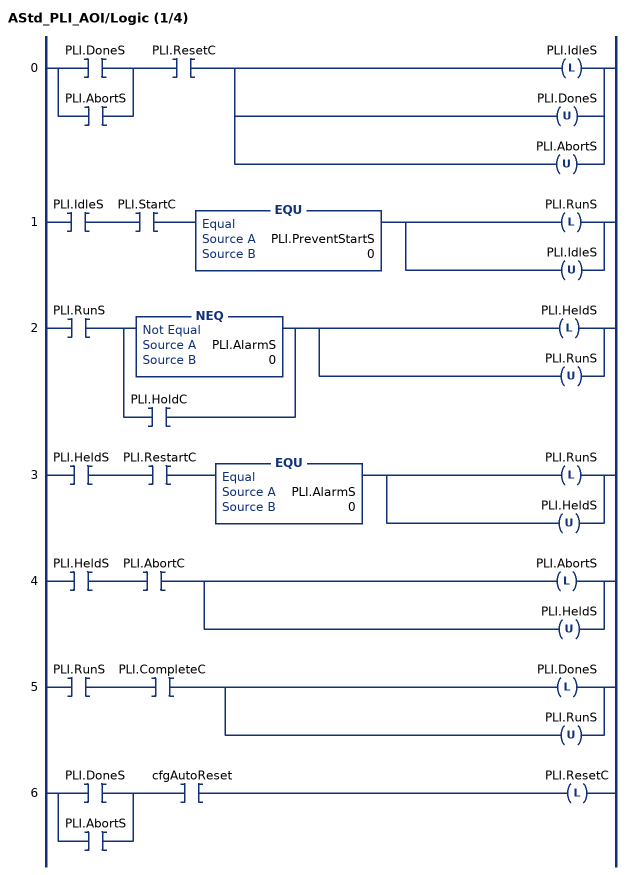
   0: [XIC(PLI.DoneS) ,XIC(PLI.AbortS) ]XIC(PLI.ResetC)[OTL(PLI.IdleS) ,OTU(PLI.DoneS) ,OTU(PLI.AbortS) ];
   1: XIC(PLI.IdleS)XIC(PLI.StartC)EQU(PLI.PreventStartS,0)[OTL(PLI.RunS) ,OTU(PLI.IdleS) ];
   2: XIC(PLI.RunS)[NEQ(PLI.AlarmS,0) ,XIC(PLI.HoldC) ][OTL(PLI.HeldS) ,OTU(PLI.RunS) ];
   3: XIC(PLI.HeldS)XIC(PLI.RestartC)EQU(PLI.AlarmS,0)[OTL(PLI.RunS) ,OTU(PLI.HeldS) ];
   4: XIC(PLI.HeldS)XIC(PLI.AbortC)[OTL(PLI.AbortS) ,OTU(PLI.HeldS) ];
   5: XIC(PLI.RunS)XIC(PLI.CompleteC)[OTL(PLI.DoneS) ,OTU(PLI.RunS) ];
   6: [XIC(PLI.DoneS) ,XIC(PLI.AbortS) ]XIC(cfgAutoReset)OTL(PLI.ResetC);
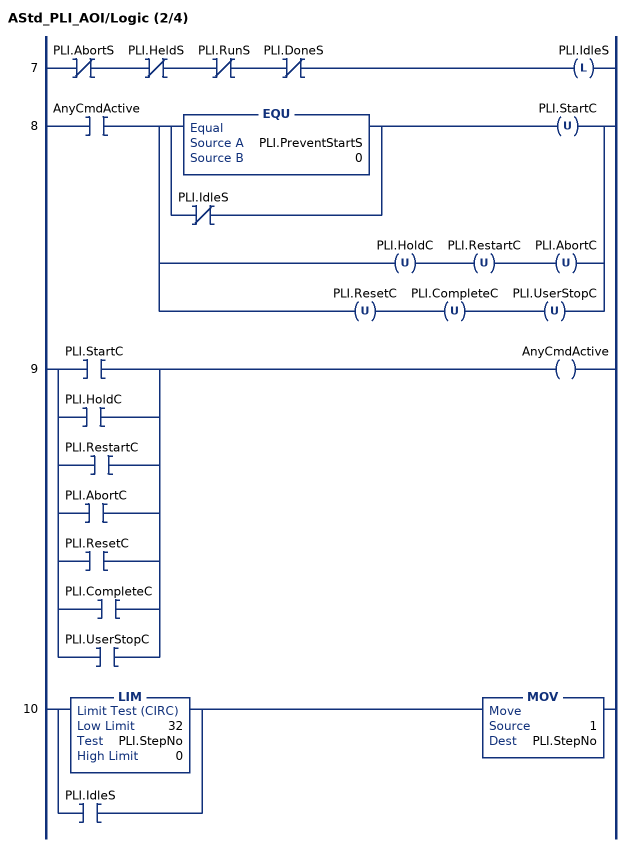
   7: XIO(PLI.AbortS)XIO(PLI.HeldS)XIO(PLI.RunS)XIO(PLI.DoneS)OTL(PLI.IdleS);
   8: XIC(AnyCmdActive)[[EQU(PLI.PreventStartS,0) ,XIO(PLI.IdleS) ] OTU(PLI.StartC) ,OTU(PLI.HoldC) OTU(PLI.RestartC) OTU(PLI.AbortC) ,OTU(PLI.ResetC) OTU(PLI.CompleteC) OTU(PLI.UserStopC) ];
   9: [XIC(PLI.StartC) ,XIC(PLI.HoldC) ,XIC(PLI.RestartC) ,XIC(PLI.AbortC) ,XIC(PLI.ResetC) ,XIC(PLI.CompleteC) ,XIC(PLI.UserStopC) ]OTE(AnyCmdActive);
   10: [LIM(32,PLI.StepNo,0) ,XIC(PLI.IdleS) ]MOV(1,PLI.StepNo);
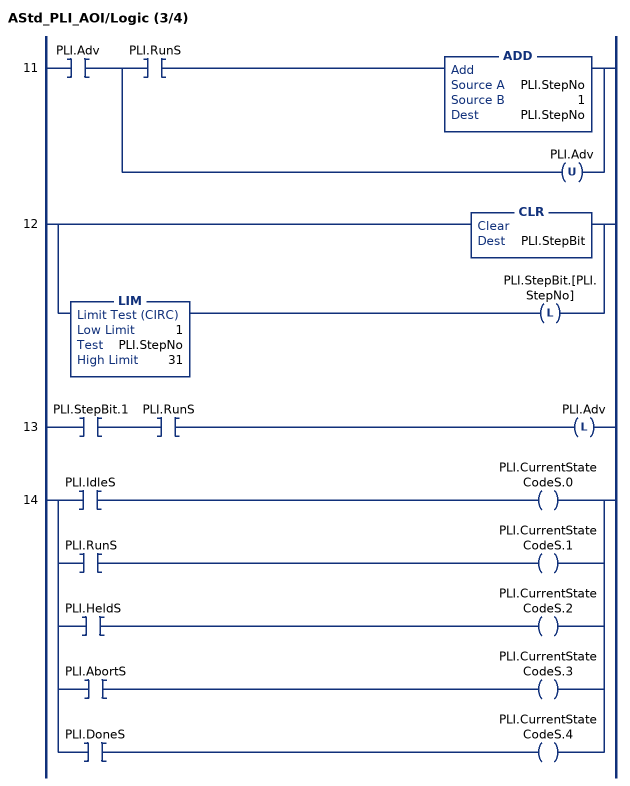
   11: XIC(PLI.Adv)[XIC(PLI.RunS) ADD(PLI.StepNo,1,PLI.StepNo) ,OTU(PLI.Adv) ];
   12: [CLR(PLI.StepBit) ,LIM(1,PLI.StepNo,31) OTL(PLI.StepBit.[PLI.StepNo]) ];
   13: XIC(PLI.StepBit.1)XIC(PLI.RunS)OTL(PLI.Adv);
   14: [XIC(PLI.IdleS) OTE(PLI.CurrentStateCodeS.0) ,XIC(PLI.RunS) OTE(PLI.CurrentStateCodeS.1) ,XIC(PLI.HeldS) OTE(PLI.CurrentStateCodeS.2) ,XIC(PLI.AbortS) OTE(PLI.CurrentStateCodeS.3) ,XIC(PLI.DoneS) OTE(PLI.CurrentStateCodeS.4) ];
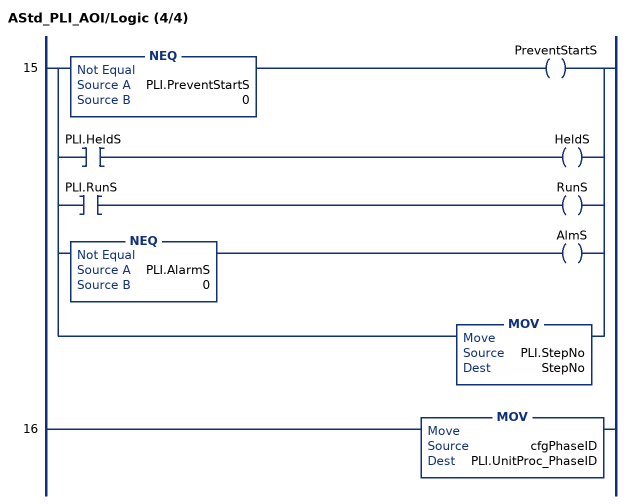
   15: [NEQ(PLI.PreventStartS,0) OTE(PreventStartS) ,XIC(PLI.HeldS) OTE(HeldS) ,XIC(PLI.RunS) OTE(RunS) ,NEQ(PLI.AlarmS,0) OTE(AlmS) ,MOV(PLI.StepNo,StepNo) ];
   16: MOV(cfgPhaseID,PLI.UnitProc_PhaseID);
END_ROUTINE
END_ADD_ON_INSTRUCTION
